# EPICS substitutions: pymcaApp/Db/pymca.substitutions
file File.template
{
pattern {P,R}
{  HB3, : }
}

file StatsInfo.template
{
pattern {P,R}
{  HB3, : }
}
